// TIA Portal V18 export
FUNCTION_BLOCK "LGasp_ProdLunghezze"   // FB10309, LAD
{ S7_Optimized_Access := 'TRUE' }
VERSION : 0.1
// stored: AutoNumber false, IsIECCheckEnabled false, IsRetainMemResEnabled false, MemoryReserve 100, SetENOAutomatically false, UDAEnableTagReadback false
   VAR_INPUT
      i_lista_compilata { ExternalAccessible := 'False'; ExternalVisible := 'False'; ExternalWritable := 'False'} : Bool;   // azzerabuffer riordino e comincia a riordinare
      i_reset { ExternalAccessible := 'False'; ExternalVisible := 'False'; ExternalWritable := 'False'} : Bool;
      i_richTrasfListaPrd { ExternalAccessible := 'False'; ExternalVisible := 'False'; ExternalWritable := 'False'} : Bool;   // richiesta trasferimento lista produzione da PC
      i_correttore { ExternalAccessible := 'False'; ExternalVisible := 'False'; ExternalWritable := 'False'} : LReal := 1.0;
   END_VAR
   VAR_OUTPUT
      o_DatiProdOK { ExternalAccessible := 'False'; ExternalVisible := 'False'; ExternalWritable := 'False'} : Bool;   // Lunghezze presenti in tabella di produzione
      o_OkTrasfListaPrd { ExternalAccessible := 'False'; ExternalVisible := 'False'; ExternalWritable := 'False'} : Bool;
      o_AlmFinePezzi { ExternalAccessible := 'False'; ExternalVisible := 'False'; ExternalWritable := 'False'} : Bool;
      o_LunghezzaAttuale { ExternalAccessible := 'False'; ExternalVisible := 'False'; ExternalWritable := 'False'} : LReal;   // Lunghezza pezzo attuale [mm]
      o_LunghezzaSuccessiva { ExternalAccessible := 'False'; ExternalVisible := 'False'; ExternalWritable := 'False'} : LReal;   // Lunghezza pezzo successivo [mm]
      o_MaterialeNecessario : LReal;   // Materiale necessario alla lista di produzione [mm]
   END_VAR
   VAR_IN_OUT
      io_PezzoEseguito { ExternalAccessible := 'False'; ExternalVisible := 'False'; ExternalWritable := 'False'} : Bool;   // cancella quota in lavoro
      io_cancella_pezzi { ExternalAccessible := 'False'; ExternalVisible := 'False'; ExternalWritable := 'False'} : Bool;   // cmdbool00[8]
      io_cancellazioneTotale { ExternalAccessible := 'False'; ExternalVisible := 'False'; ExternalWritable := 'False'} : Bool;   // cmdbool00[11]
      io_rich_nuovo_trasferimento { ExternalAccessible := 'False'; ExternalVisible := 'False'; ExternalWritable := 'False'} : Bool;   // richiesta nuovo trasferimento all'avvio
      io_ListaProduzionePC : Array[1.."NumRigheProduzione"] of "LGasp_typeRigaProdfromPC";
      io_myprodfromPC : Array[1.."NumRigheProduzione"] of "LGasp_typeRigaProdfromPC";
      io_myprodfromPLC : Array[1.."NumRigheProduzione"] of "LGasp_typeRigaProdfromPLC";
      io_myprodfromPCupdate : Array[1.."NumRigheProduzione"] of DInt;
      io_QuotePunzonatura : Array[1.."NumQuotePunzonatura"] of "LGasp_typeBufferQuote";
      io_StoricoRigheProdEliminate : Array[1.."NumRigheProduzione"] of "LGasp_typeRigheEliminate";
      io_ListaProfila : "LGasp_typeHMI_ListaProf";
   END_VAR
   VAR RETAIN
      s_lista_compilata_old { ExternalAccessible := 'False'; ExternalVisible := 'False'; ExternalWritable := 'False'} : Bool;
      s_inserire_pezzi_in_lista { ExternalAccessible := 'False'; ExternalVisible := 'False'; ExternalWritable := 'False'} : Bool;   // inserire pezzi in lista produzione
   END_VAR
   VAR
      s_firstScan_Done { ExternalAccessible := 'False'; ExternalVisible := 'False'; ExternalWritable := 'False'} : Bool;   // NON RITENTIVA
      s_CambioRigaProduzione { ExternalAccessible := 'False'; ExternalVisible := 'False'; ExternalWritable := 'False'} : Bool;   // Cambio riga di produzione
      s_ListaProduzione_ID_old { ExternalAccessible := 'False'; ExternalVisible := 'False'; ExternalWritable := 'False'} : Array[1.."NumRigheProduzione"] of DInt;
      s_index_0 { ExternalAccessible := 'False'; ExternalVisible := 'False'; ExternalWritable := 'False'} : DInt;
      s_index_1 { ExternalAccessible := 'False'; ExternalVisible := 'False'; ExternalWritable := 'False'} : DInt;
      s_index_2 { ExternalAccessible := 'False'; ExternalVisible := 'False'; ExternalWritable := 'False'} : DInt;
      s_index_3 { ExternalAccessible := 'False'; ExternalVisible := 'False'; ExternalWritable := 'False'} : DInt;
      s_index_4 { ExternalAccessible := 'False'; ExternalVisible := 'False'; ExternalWritable := 'False'} : DInt;
      s_index_5 { ExternalAccessible := 'False'; ExternalVisible := 'False'; ExternalWritable := 'False'} : DInt;
      s_index_6 { ExternalAccessible := 'False'; ExternalVisible := 'False'; ExternalWritable := 'False'} : DInt;
      s_index_7 { ExternalAccessible := 'False'; ExternalVisible := 'False'; ExternalWritable := 'False'} : DInt;
   END_VAR
   VAR RETAIN
      s_RigaProduzione_in_lavoro { ExternalAccessible := 'False'; ExternalVisible := 'False'; ExternalWritable := 'False'} : DInt;   // Indice riga di produzione in lavoro
   END_VAR
   VAR
      s_QuotaNULL { ExternalAccessible := 'False'; ExternalVisible := 'False'; ExternalWritable := 'False'} : "LGasp_typeQuota";   // tipo dato NULL
      s_BufferQuotaNULL { ExternalAccessible := 'False'; ExternalVisible := 'False'; ExternalWritable := 'False'} : "LGasp_typeBufferQuote";   // tipo dato NULL
      s_RigaProduzioneNULL { ExternalAccessible := 'False'; ExternalVisible := 'False'; ExternalWritable := 'False'} : "LGasp_typeRigaProdfromPC";   // tipo dato NULL
      s_mem_trasf_lista_da_PC { ExternalAccessible := 'False'; ExternalVisible := 'False'; ExternalWritable := 'False'} : Bool;
   END_VAR
   VAR RETAIN
      s_ID_righe_produzione { ExternalAccessible := 'False'; ExternalVisible := 'False'; ExternalWritable := 'False'} : Array[1.."NumRigheProduzione"] of DInt;
      s_count { ExternalAccessible := 'False'; ExternalVisible := 'False'; ExternalWritable := 'False'} : DInt;
   END_VAR
   VAR
      FP_PreFine { ExternalAccessible := 'False'; ExternalVisible := 'False'; ExternalWritable := 'False'} : R_TRIG;
      s_MaterialeNecessario { ExternalAccessible := 'False'; ExternalVisible := 'False'; ExternalWritable := 'False'} : Array[1.."NumRigheProduzione"] of LReal;
      s_appMaterialeNec { ExternalAccessible := 'False'; ExternalVisible := 'False'; ExternalWritable := 'False'} : LReal;
      s_primoTrasferimentoEseguito { ExternalAccessible := 'False'; ExternalVisible := 'False'; ExternalWritable := 'False'} : Bool;
   END_VAR
   VAR_TEMP   // added for the SCL form of the ladder/FBD networks
      _w1 : Bool;
   END_VAR
BEGIN

REGION Network 1 (SCL): Descrizione
   //================================================================================
   // Gasparini Spa
   //--------------------------------------------------------------------------------
   // Libreria: LGasp_ProdLunghezze
   // Funzionalità: Funzione globale per gestione riordino quote
   // Commessa in cui è stata testata: YYXXNNNNN
   // Programmatore di riferimento per test: XXXXXX
   //--------------------------------------------------------------------------------
   // Change log table:
   // Versione Data        Autore          Modifiche
   // 01.00.05 08/04/2021  Lcg             Rilascio funzione testata la prima volta su micron 305
   // 02.00.00 10.12.2021  Enzo            Aggiunto popolamento lista profila anche quando si ha solo lista lunghezza *210100057*
   // 02.00.01 01.04.2022  Lcg             Aggiunti due parametri di uscita, lunghezza successiva e quantità totale di materiale necessario 
   //                                      per eseguire la produzione impostata
   // 02.00.02 28.09.2022  Lcg             Inserito numero del pezzo in lista profila (Bito 210100099)
   // 02.00.03 06.10.2022  Lcg             Inserita la gestione delle nuove variabili "opzioni" personalizzabili a seconda della macchina (Bito 210100099)
   // 02.00.04 14/03/2023  Lcg             Corretto errore che all'avvio azzerava i pezzi fatti dopo uno snapshot di L1_prd (22010003)
   // 02.00.05 17/03/2023  Lcg             Corretto errore "Allarme fine pezzi" all'accensione, si attende il primo trasferimento.  
   //-------------------------------------------------------------------------------
   //================================================================================
END_REGION

REGION Network 2 (SCL): Appoggio Produzione dal PC sulla produzione del PLC


   IF #i_richTrasfListaPrd THEN
       #s_mem_trasf_lista_da_PC := TRUE;
   END_IF;

   IF NOT #i_richTrasfListaPrd AND #s_mem_trasf_lista_da_PC THEN
       #s_mem_trasf_lista_da_PC := FALSE;
       #io_myprodfromPC :=  #io_ListaProduzionePC;
   END_IF;
END_REGION

REGION Network 3 (SCL): Cancellazione totale
       IF #io_cancellazioneTotale THEN

           //cancella quote punzonatura
           FOR #s_index_1 := 1 TO "NumQuotePunzonatura" DO // Statement section IF
               #io_QuotePunzonatura[#s_index_1] := #s_BufferQuotaNULL;
           END_FOR;

           //cancello tutto
           FOR #s_index_1 := 1 TO "NumRigheProduzione" DO
               #io_myprodfromPLC[#s_index_1].pzinseritinelriordinoquote := 0;
               #io_myprodfromPLC[#s_index_1].pzfatti := 0;

               #io_myprodfromPC[#s_index_1].ID := 0;
               #io_myprodfromPC[#s_index_1].piecestodo := 0;
               #io_myprodfromPC[#s_index_1].tipoarticolo := 0;

           END_FOR;

           #io_cancellazioneTotale := false;
       END_IF;
END_REGION

REGION Network 4 (SCL): Riga di produzione in lavoro
   FOR #s_index_1 := 1 TO "NumRigheProduzione" DO
       IF #io_myprodfromPLC[#s_index_1].pzfatti < #io_myprodfromPC[#s_index_1].piecestodo THEN
           #s_RigaProduzione_in_lavoro := #s_index_1;
           EXIT;
       END_IF;
   END_FOR;
END_REGION

REGION Network 5 (SCL): Lavorazione eseguita
   // comando pezzo eseguito
   IF #io_PezzoEseguito THEN

       // incremento pezzi fatti
       #io_myprodfromPLC[#s_RigaProduzione_in_lavoro].pzfatti := #io_myprodfromPLC[#s_RigaProduzione_in_lavoro].pzfatti + 1;

       // Aggiorno lista profila
       IF #io_ListaProfila.abilitata THEN
           // Popolo i campi del pezzo da inserire
           #io_ListaProfila.pezzo_fatto.ID := #io_myprodfromPC[#s_RigaProduzione_in_lavoro].ID;
           #io_ListaProfila.pezzo_fatto.lenght := #io_myprodfromPC[#s_RigaProduzione_in_lavoro].article.general.lenght;
           #io_ListaProfila.pezzo_fatto.cutoffset := #io_myprodfromPC[#s_RigaProduzione_in_lavoro].article.general.cutoffset;
           #io_ListaProfila.pezzo_fatto.wastepiece := false;

           #io_ListaProfila.pezzo_fatto.options := #io_myprodfromPC[#s_RigaProduzione_in_lavoro].article.general.options;
           #io_ListaProfila.pezzo_fatto.options_dint := #io_myprodfromPC[#s_RigaProduzione_in_lavoro].article.general.options_dint;
           #io_ListaProfila.pezzo_fatto.options_lreal := #io_myprodfromPC[#s_RigaProduzione_in_lavoro].article.general.options_lreal;
           #io_ListaProfila.pezzo_fatto.options_str:= #io_myprodfromPC[#s_RigaProduzione_in_lavoro].article.general.options_str;

           //numerpo del pezzo per lista profila
           #io_ListaProfila.pezzo_fatto.NumeroPezzo := #io_myprodfromPLC[#s_RigaProduzione_in_lavoro].pzfatti;

           // Inserimento pezzo in profila
           #io_ListaProfila.io_inserisci_pzo_buono := true;

       END_IF;


       //aggiorno anche pezzi in riordino per bloccare le modifiche nel PC della riga attualmente in lavoro in pagina di produzione
       IF #io_myprodfromPLC[#s_RigaProduzione_in_lavoro].pzfatti < #io_myprodfromPC[#s_RigaProduzione_in_lavoro].piecestodo THEN
           #io_myprodfromPLC[#s_RigaProduzione_in_lavoro].pzinseritinelriordinoquote := #io_myprodfromPLC[#s_RigaProduzione_in_lavoro].pzfatti + 1;
       END_IF;

       //se nella riga c'è un pezzo solo pezzi in riordino uguale a pezzi fatti
       IF #io_myprodfromPLC[#s_RigaProduzione_in_lavoro].pzfatti = #io_myprodfromPC[#s_RigaProduzione_in_lavoro].piecestodo AND #io_myprodfromPC[#s_RigaProduzione_in_lavoro].piecestodo = 1 THEN
           #io_myprodfromPLC[#s_RigaProduzione_in_lavoro].pzinseritinelriordinoquote := #io_myprodfromPLC[#s_RigaProduzione_in_lavoro].pzfatti;
       END_IF;

       // fine
       #io_PezzoEseguito := false;

   END_IF;
END_REGION

REGION Network 6: Quote ok
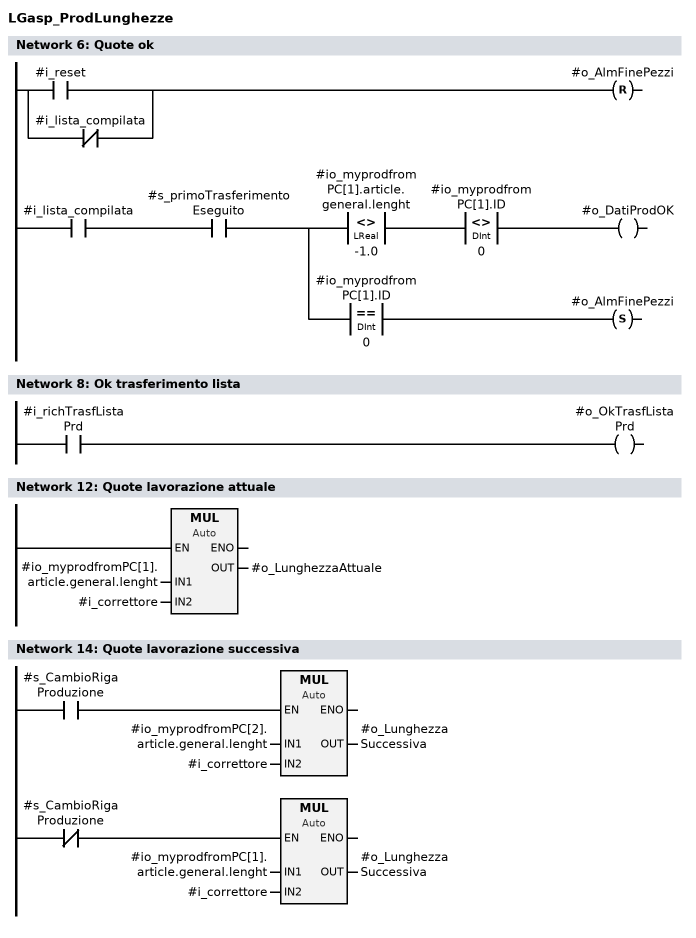
   RUNG wire#powerrail
      Contact( #i_reset )
      wire#w1
      R_Coil( #o_AlmFinePezzi )
   END_RUNG
   RUNG wire#powerrail
      I_Contact( #i_lista_compilata )
   END_RUNG wire#w1
   RUNG wire#powerrail
      Contact( #i_lista_compilata )
      Contact( #s_primoTrasferimentoEseguito )
      wire#w2
      { S7_Templates := "SrcType := LReal" } NE_Contact(in1 := #io_myprodfromPC[1].article.general.lenght, in2 := -1.0)
      { S7_Templates := "SrcType := DInt" } NE_Contact(in1 := #io_myprodfromPC[1].ID, in2 := 0)
      Coil( #o_DatiProdOK )
   END_RUNG
   RUNG wire#w2
      { S7_Templates := "SrcType := DInt" } EQ_Contact(in1 := #io_myprodfromPC[1].ID, in2 := 0)
      S_Coil( #o_AlmFinePezzi )
   END_RUNG
   // the same network as SCL:
   IF #i_reset OR NOT #i_lista_compilata THEN #o_AlmFinePezzi := FALSE; END_IF;
   #_w1 := #i_lista_compilata AND #s_primoTrasferimentoEseguito;
   #o_DatiProdOK := #_w1 AND (#io_myprodfromPC[1].article.general.lenght <> (-1.0)) AND (#io_myprodfromPC[1].ID <> 0);
   IF #_w1 AND (#io_myprodfromPC[1].ID = 0) THEN #o_AlmFinePezzi := TRUE; END_IF;
END_REGION

REGION Network 7 (SCL): Elimina righe terminate (attenzione le elimino solo da parte PLC )
   IF NOT #s_mem_trasf_lista_da_PC AND #s_primoTrasferimentoEseguito THEN

       IF (#io_myprodfromPLC[1].pzfatti >= #io_myprodfromPC[1].piecestodo) AND (#io_myprodfromPC[1].piecestodo > 0) THEN


           //salvataggio ID e pezzi fatti della riga appena completata: serve al PC per impostare correttamente i pezzi fatti
           //nelle righe eliminate
           //spostamento delle righe 
           FOR #s_index_5 := 0 TO "NumRigheProduzione" - 2 DO
               #io_StoricoRigheProdEliminate[NumRigheProduzione - #s_index_5] := #io_StoricoRigheProdEliminate[NumRigheProduzione - #s_index_5 - 1];
           END_FOR;

           //salvataggio ID e pezzi fatti prima di eliminare la riga di produzione
           #io_StoricoRigheProdEliminate[1].ID := #io_myprodfromPC[1].ID;
           #io_StoricoRigheProdEliminate[1].pzfatti := #io_myprodfromPLC[1].pzfatti;

           //cancella pezzi fatti
           #io_myprodfromPLC[1].pzfatti := 0;

           //salvataggio nuovi dati

           //sposta le righe di produzione
           FOR #s_index_5 := 1 TO "NumRigheProduzione" - 1 DO
               #io_myprodfromPC[#s_index_5] := #io_myprodfromPC[#s_index_5 + 1];
               #io_myprodfromPLC[#s_index_5] := #io_myprodfromPLC[#s_index_5 + 1];
           END_FOR;

           #io_myprodfromPC[NumRigheProduzione] := #s_RigaProduzioneNULL;

       END_IF;
   END_IF;
END_REGION

REGION Network 8: Ok trasferimento lista
   RUNG wire#powerrail
      Contact( #i_richTrasfListaPrd )
      Coil( #o_OkTrasfListaPrd )
   END_RUNG
   // the same network as SCL:
   #o_OkTrasfListaPrd := #i_richTrasfListaPrd;
END_REGION

REGION Network 9 (SCL): Cancella pezzi fatti
   IF NOT #i_lista_compilata AND #io_cancella_pezzi THEN
       FOR #s_index_7 := 1 TO "NumRigheProduzione" DO
           #io_myprodfromPLC[#s_index_7].pzfatti := 0;
           #io_myprodfromPLC[#s_index_7].pzinseritinelriordinoquote := 0;
       END_FOR;
   END_IF;

   #io_cancella_pezzi := false;
END_REGION

REGION Network 10 (SCL): Aggiornamento pezzi da fare durante la marcia
   // Controllo se sono stati modificati i pezzi da fare in pagina di produzione e aggiorno le righe di produzione con i nuovi pezzi
       FOR #s_index_7 := 1 TO "NumRigheProduzione" DO

           IF #io_myprodfromPCupdate[#s_index_7] > 0 AND #io_myprodfromPCupdate[#s_index_7] > #io_myprodfromPLC[#s_index_7].pzinseritinelriordinoquote THEN
               #io_myprodfromPC[#s_index_7].piecestodo := #io_myprodfromPCupdate[#s_index_7];
           END_IF;
           #io_myprodfromPCupdate[#s_index_7] := 0;

       END_FOR;
END_REGION

REGION Network 11 (SCL): Memoria ID prima riga per riallineamento all'accensione
   IF NOT #s_firstScan_Done THEN

       FOR #s_index_0 := 1 TO "NumRigheProduzione" DO
           #io_myprodfromPC[#s_index_0].ID := #s_ID_righe_produzione[#s_index_0];
       END_FOR;

       #io_rich_nuovo_trasferimento := true;
       #s_firstScan_Done := true;

   END_IF;

   IF #s_firstScan_Done AND NOT #io_rich_nuovo_trasferimento THEN
       FOR #s_index_0 := 1 TO "NumRigheProduzione" DO
           #s_ID_righe_produzione[#s_index_0] := #io_myprodfromPC[#s_index_0].ID;
       END_FOR;
       #s_primoTrasferimentoEseguito := true;
   END_IF;
END_REGION

REGION Network 12: Quote lavorazione attuale
   RUNG wire#powerrail
      Mul(in1 := #io_myprodfromPC[1].article.general.lenght, in2 := #i_correttore, out => #o_LunghezzaAttuale)
   END_RUNG
   // the same network as SCL:
   #o_LunghezzaAttuale := #io_myprodfromPC[1].article.general.lenght * #i_correttore;
END_REGION

REGION Network 13 (SCL): calcolo cambio riga
   IF #io_myprodfromPLC[1].pzfatti > #io_myprodfromPC[1].piecestodo - 2 THEN
       #s_CambioRigaProduzione := TRUE;
   ELSE
       #s_CambioRigaProduzione := FALSE;
   END_IF;
END_REGION

REGION Network 14: Quote lavorazione successiva
   RUNG wire#powerrail
      Contact( #s_CambioRigaProduzione )
      Mul(in1 := #io_myprodfromPC[2].article.general.lenght, in2 := #i_correttore, out => #o_LunghezzaSuccessiva)
   END_RUNG
   RUNG wire#powerrail
      I_Contact( #s_CambioRigaProduzione )
      Mul(in1 := #io_myprodfromPC[1].article.general.lenght, in2 := #i_correttore, out => #o_LunghezzaSuccessiva)
   END_RUNG
   // the same network as SCL:
   IF #s_CambioRigaProduzione THEN
       #o_LunghezzaSuccessiva := #io_myprodfromPC[2].article.general.lenght * #i_correttore;
   END_IF;
   IF NOT #s_CambioRigaProduzione THEN
       #o_LunghezzaSuccessiva := #io_myprodfromPC[1].article.general.lenght * #i_correttore;
   END_IF;
END_REGION

REGION Network 15 (SCL): lamiera totale necessaria per eseguire la produzione
       #s_appMaterialeNec := 0;
       FOR #s_index_0 := 1 TO "NumRigheProduzione" DO
           #s_MaterialeNecessario[#s_index_0] := ((#io_myprodfromPC[#s_index_0].piecestodo - #io_myprodfromPLC[#s_index_0].pzfatti) * #io_myprodfromPC[#s_index_0].article.general.lenght);
           #s_appMaterialeNec := #s_appMaterialeNec + #s_MaterialeNecessario[#s_index_0];
           IF #s_index_0 = "NumRigheProduzione" THEN
               #o_MaterialeNecessario := #s_appMaterialeNec;
           END_IF;
       END_FOR;
END_REGION
END_FUNCTION_BLOCK
